(* IEC 61131-3 sources: stverif/testfiles/Blackbox/src/rule2, 1 file *)

(* ---- rule2.st ---- *)
PROGRAM _CYCLIC
	IF a > b THEN
		c := a;
	ELSE
		c := b;
	END_IF
END_PROGRAM
